{attribute 'linkalways'} 
{attribute 'no_explicit_call' := 'This FB is a CLASS and must be accessed using methods or properties'}
{attribute 'enable_dynamic_creation'}
FUNCTION_BLOCK _ETcVnDrawShape EXTENDS EnumDatatypeBase
VAR
	localData : ETcVnDrawShape;
	activeData : REFERENCE TO ETcVnDrawShape;
	enumBaseDatatype : _DINT(localData);
END_VAR

METHOD PRIVATE AddLocalEnumeration
VAR_INPUT
	Enumeration : T_MAXSTRING;
	Value : ETcVnDrawShape;
END_VAR
AddEnumeration(Enumeration, Value);
END_METHOD

PROPERTY PUBLIC Address : PVOID
GET
Address := ADR(activeData);
END_GET
END_PROPERTY

METHOD PUBLIC ClearReference
VAR_INPUT
END_VAR
activeData REF= localData;
SetBaseDatatypeReference();
END_METHOD

METHOD PUBLIC Clone : I_Datatype
VAR
    pClone : POINTER TO _ETcVnDrawShape;
END_VAR
pClone := __NEW(_ETcVnDrawShape(InitialValue := Value));
Clone := pClone^;
END_METHOD

METHOD FB_init : BOOL
VAR_INPUT
	bInitRetains : BOOL; // if TRUE, the retain variables are initialized (warm start / cold start)
	bInCopyCode : BOOL;  // if TRUE, the instance afterwards gets moved into the copy code (online change)
	InitialValue : ETcVnDrawShape;
END_VAR
localData := InitialValue;
AddBaseDatatype(enumBaseDatatype);
ClearReference();

AddLocalEnumeration('TCVN_DS_RANDOM', ETcVnDrawShape.TCVN_DS_RANDOM);
AddLocalEnumeration('TCVN_DS_CIRCLE', ETcVnDrawShape.TCVN_DS_CIRCLE);
AddLocalEnumeration('TCVN_DS_SQUARE', ETcVnDrawShape.TCVN_DS_SQUARE);
AddLocalEnumeration('TCVN_DS_PLUS', ETcVnDrawShape.TCVN_DS_PLUS);
AddLocalEnumeration('TCVN_DS_X', ETcVnDrawShape.TCVN_DS_X);
AddLocalEnumeration('TCVN_DS_DIAMOND', ETcVnDrawShape.TCVN_DS_DIAMOND);
AddLocalEnumeration('TCVN_DS_MAX', ETcVnDrawShape.TCVN_DS_MAX);
END_METHOD

PROPERTY PUBLIC Identifier : T_MAXSTRING
GET
Identifier := 'ETcVnDrawShape';
END_GET
END_PROPERTY

METHOD IsEnumeratorValueEqual : BOOL
VAR_INPUT
	Enumerator : I_KeyValueForwardEnumerator;
END_VAR
VAR
	storedValue : ETcVnDrawShape;
END_VAR
IF NOT Enumerator.TryGet(storedValue) THEN
	RETURN;
END_IF

IsEnumeratorValueEqual := storedValue = activeData;
END_METHOD

METHOD PUBLIC MakeReferenceTo
VAR_INPUT
	ReferenceTarget : REFERENCE TO ETcVnDrawShape;
END_VAR
activeData REF= ReferenceTarget;
SetBaseDatatypeReference();
END_METHOD

METHOD PROTECTED SetBaseDatatypeReference
VAR_INPUT
END_VAR
enumBaseDatatype.MakeReferenceTo(activeData);
END_METHOD

PROPERTY PUBLIC Size : UDINT
GET
Size := SIZEOF(activeData);
END_GET
END_PROPERTY

METHOD TryMakeReferenceTo : BOOL
VAR_INPUT
	Target : I_Datatype;
END_VAR
VAR
	pTargetData : POINTER TO ETcVnDrawShape;
END_VAR
IF NOT IsEquivalentTo(Target) THEN
	RETURN;
END_IF

pTargetData := Target.Address;
activeData REF= pTargetData^;
SetBaseDatatypeReference();
TryMakeReferenceTo := TRUE;
END_METHOD

PROPERTY PUBLIC Value : ETcVnDrawShape
GET
Value := activeData;
END_GET
SET
activeData := Value;
END_SET
END_PROPERTY

END_FUNCTION_BLOCK

(* stored: Version 1.1.0.1, ProductVersion 3.1.4024.13
   POU _ETcVnDrawShape: Id {22f1166e-ac14-0deb-11be-9b1524b9543f}, SpecialFunc None
   Folder Core: Id {5bbf99a7-04f5-0fae-114e-45bfe15f71ee}
   Folder Protected: Id {8c66a33d-f95c-0ba8-1852-91f53622bb5d}
   Folder Customize: Id {25197707-f455-02c9-3fcb-c3527a9b2e68}
   Folder Constructor: Id {77f505a2-38f6-0391-2134-7e69d6f95644}
   Folder Private: Id {5c5ee1e5-e974-0ccb-2010-29ac0056f2e1}
   Folder Protected: Id {3fe08415-f3ce-03a4-2e8a-1e1356caa7ed}
   Method AddLocalEnumeration: Id {f47a731f-62f8-0990-3589-ca6e4ef3b73c}
   Property Address: Id {d329098f-fba2-036e-2b92-36ac98716474}
   Get Get: Id {1c0e7b7d-4e9f-0a3f-306f-7ced7eca348c}
   Method ClearReference: Id {aea813ef-b355-0538-3557-fc6ba2639899}
   Method Clone: Id {aefe02a6-51d5-0dd1-09d2-dc31c4ff304c}
   Method FB_init: Id {9005c7fc-9d24-0d41-3d84-85e49f0ef410}
   Property Identifier: Id {c1b73de9-c6a6-06d0-0b7a-1b0d958afc80}
   Get Get: Id {e35223b5-4c9f-0249-0c8f-045b12ccf693}
   Method IsEnumeratorValueEqual: Id {12c61453-a37c-00fe-2ae2-da842e6c9db9}
   Method MakeReferenceTo: Id {b1616947-7dc3-0411-0cf2-ac607ea3f913}
   Method SetBaseDatatypeReference: Id {3ae92a96-a4d7-01e5-22aa-cc2a529cf6b3}
   Property Size: Id {10927b86-2fc7-0561-2f79-77d881851930}
   Get Get: Id {18173c76-a6a4-0a1a-1e22-1cf8574e98d3}
   Method TryMakeReferenceTo: Id {7dae5580-98ea-0a80-1a6a-8bfaa6a7f7b2}
   Property Value: Id {b323c504-7ed2-0340-2a16-6f03a32d7f82}
   Get Get: Id {4c525c40-cbcb-0ed6-1e56-3c6e810c6d26}
   Set Set: Id {434829e7-570c-048d-077e-fe99969dd354} *)
